Fanuc KAREL source: kb00015.KL

PROGRAM KB00015
%NOLOCKGROUP
VAR
P1 : STRING[80];P2:INTEGER
BEGIN
--
P1='A'
P2=1
CALL_PROG(P1,P2)
END KB00015
